// SIMATIC S7-200 project (STEP 7-Micro/WIN), CPU 221 REL 01.10

SYMBOL_TABLE USER1
Mode             I0.0
Reset            I0.1
Stopp            I0.2
Xanh_1           Q0.0
Vang_1           Q0.1
Do_1             Q0.2
Xanh_2           Q0.3
Vang_2           Q0.4
Do_2             Q0.5
DEN_CD1          Q1.0
DEN_CD2          Q1.1
END_SYMBOL_TABLE

ORGANIZATION_BLOCK MAIN:OB1
TITLE=PROGRAM COMMENTS
BEGIN
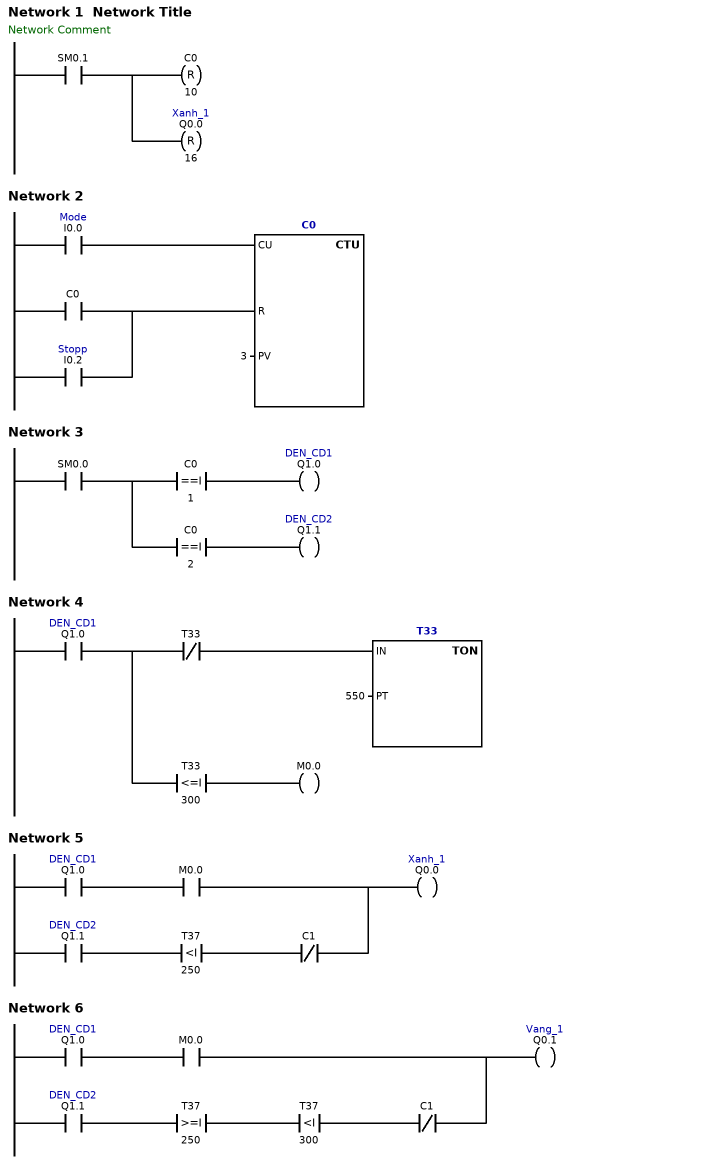
Network 1 // Network Title
// Network Comment
LD     SM0.1
R      C0, 10
R      Xanh_1:Q0.0, 16
Network 2
LD     Mode:I0.0
LD     C0
O      Stopp:I0.2
CTU    C0, 3
Network 3
LD     SM0.0
LPS
AW=    C0, 1
=      DEN_CD1:Q1.0
LPP
AW=    C0, 2
=      DEN_CD2:Q1.1
Network 4
LD     DEN_CD1:Q1.0
LPS
AN     T33
TON    T33, 550
LPP
AW<=   T33, 300
=      M0.0
Network 5
LD     DEN_CD1:Q1.0
A      M0.0
LD     DEN_CD2:Q1.1
AW<    T37, 250
AN     C1
OLD
=      Xanh_1:Q0.0
Network 6
LD     DEN_CD1:Q1.0
A      M0.0
LD     DEN_CD2:Q1.1
AW>=   T37, 250
AW<    T37, 300
AN     C1
OLD
=      Vang_1:Q0.1
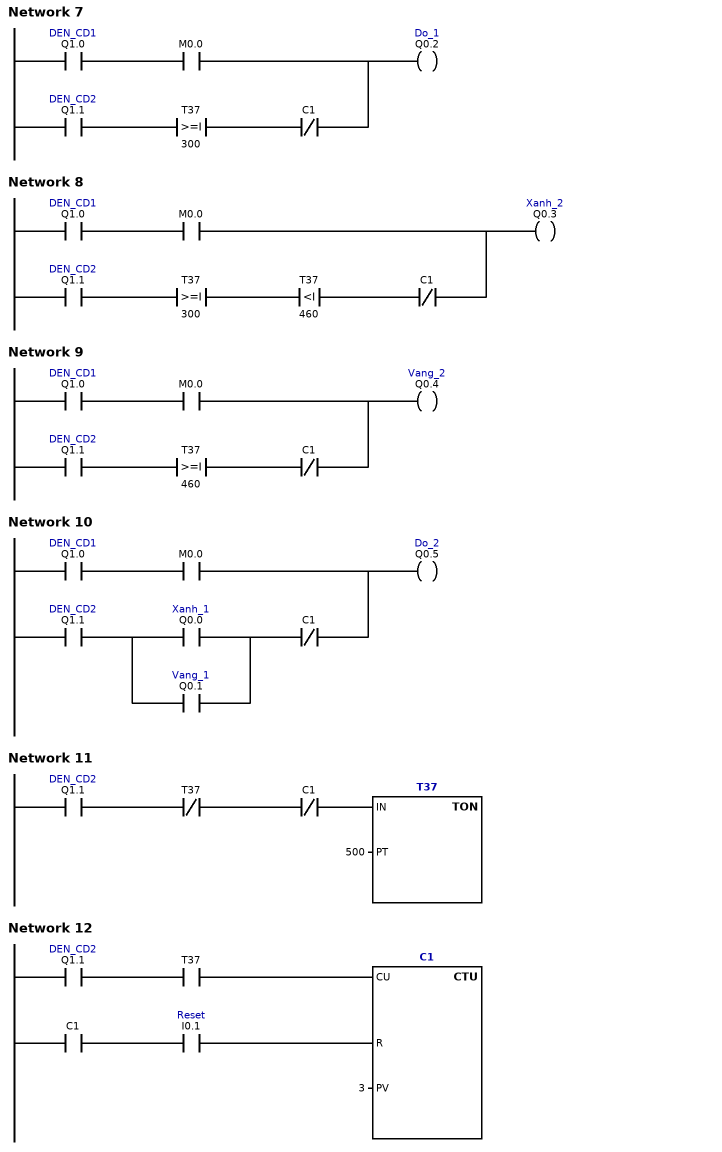
Network 7
LD     DEN_CD1:Q1.0
A      M0.0
LD     DEN_CD2:Q1.1
AW>=   T37, 300
AN     C1
OLD
=      Do_1:Q0.2
Network 8
LD     DEN_CD1:Q1.0
A      M0.0
LD     DEN_CD2:Q1.1
AW>=   T37, 300
AW<    T37, 460
AN     C1
OLD
=      Xanh_2:Q0.3
Network 9
LD     DEN_CD1:Q1.0
A      M0.0
LD     DEN_CD2:Q1.1
AW>=   T37, 460
AN     C1
OLD
=      Vang_2:Q0.4
Network 10
LD     DEN_CD1:Q1.0
A      M0.0
LD     DEN_CD2:Q1.1
LD     Xanh_1:Q0.0
O      Vang_1:Q0.1
ALD
AN     C1
OLD
=      Do_2:Q0.5
Network 11
// (network saved uncompiled; LAD cells follow)
// row 0: c0 -| |- DEN_CD2:Q1.1  c1 -|/|- T37  c2 -|/|- C1  c3 [TON T37 IN:=power@row0, PT:=500]
// row 1: c3 [box]
Network 12
LD     DEN_CD2:Q1.1
A      T37
LD     C1
A      Reset:I0.1
CTU    C1, 3
END_ORGANIZATION_BLOCK
